FUNCTION EXPN : REAL
VAR_INPUT
	X : REAL;
	N : INT;
END_VAR
VAR
	sign: BOOL;
END_VAR

(*
version 1.2	10. mar. 2009
programmer 	hugo
tested by		oscat

this function calculates X to the power of N (Y = X^N) whilke N is an integer
especially on CPU's without a floating point unit this algorythm is about 30 times faster then the IEC standard EXPT() Function

*)

sign := n.15;
N := ABS(N);
IF N.0 THEN EXPN := X; ELSE EXPN := 1.0; END_IF;
N := SHR(N,1);
WHILE N > 0 DO
   X := X * X;
   IF N.0 THEN EXPN := EXPN * X; END_IF;
   N := SHR(N,1);
END_WHILE;
IF sign THEN EXPN := 1.0 / EXPN; END_IF;



(* revision history
hm	4. dec 2007	rev 1.0
	original version

hm	22. oct. 2008	rev 1.1
	optimized code

hm	10. mar. 2009	rev 1.2
	removed nested comments
	real constants updated to new systax using dot

*)

END_FUNCTION

(* stored: Version 1.1.0.1, ProductVersion 3.1.4022.7
   POU EXPN: Id {ad8a8f99-24b4-4a18-9251-4c2905324bfa}, SpecialFunc None *)
